// Mitsubishi GX Works2 project: CydeusPlatform3   PLC: FX3U/FX3UC

TYPE ST_1SolCylinderInterface : STRUCT
  bBusy : BOOL;
  bError : BOOL;
  bDone : BOOL;
  bGoActive : BOOL;
  bReset : BOOL;
  tDelayTime : TIME;
  tTimeout : TIME;
  bAbort : BOOL;
END_STRUCT END_TYPE

TYPE ST_ServoMotorInterface : STRUCT
  bBusy : BOOL;
  bError : BOOL;
  bDone : BOOL;
  bServoEnabled : BOOL;
  bEnable : BOOL;
  bStop : BOOL;
  bAbort : BOOL;
  bReset : BOOL;
  bJogPos : BOOL;
  bJogNeg : BOOL;
  bMoveRel : BOOL;
  rMoveDist : REAL;
  rMoveVel : REAL;
  rMoveAccel : REAL;
  rJogVel : REAL;
END_STRUCT END_TYPE

// global labels: GVL_Error
VAR_GLOBAL
  arrError AT M200 : ARRAY [0..9] OF BOOL;  (* List of Current active error *)
END_VAR
VAR_GLOBAL CONSTANT
  uiNumErrMinus1 : INT := 9;  (* Maximum error minus 1 *)
END_VAR
VAR_GLOBAL
  arrMsg AT M250 : ARRAY [0..9] OF BOOL;  (* List of Current active message *)
END_VAR
VAR_GLOBAL CONSTANT
  uiNumMsgMinus1 : INT := 9;  (* Maximum message minus 1 *)
END_VAR

// global labels: GVL_Main
VAR_GLOBAL
  bAlarmTrigger : BOOL;  (* Simulating Alarm Trigger *)
  bMachineError AT M100 : BOOL;  (* Machine error *)
  bManualMode : BOOL;  (* Manual Mode on *)
  bAutoMode : BOOL;  (* Automatic Mode on *)
  bStepMode : BOOL;  (* Step Mode on *)
  bSimMode : BOOL;  (* Simulation Mode on *)
  objPunching : CL_1Sol1SenCylinder;  (* Punching object *)
  stServoMotor : ST_ServoMotorInterface;  (* Servo Motor interface struct *)
  stPunching : ST_1SolCylinderInterface;  (* Punching interface struct *)
  objServoMotor : CL_ServoMotor;  (* Servo Motor object *)
  bManualEnable : BOOL;  (* Manual Mode enabled *)
  bMachineReady AT M101 : BOOL;  (* Machine Ready *)
END_VAR

// global labels: GVL_HMI
VAR_GLOBAL
  btnInitialize AT M2 : BOOL;  (* Begin button *)
  btnAutoMode AT M4 : BOOL;  (* Automatic Mode button *)
  btnStepMode AT M5 : BOOL;  (* Step Mode button *)
  btnTest AT M7 : BOOL;  (* Test Mode button *)
  btnTestManualOn AT M8 : BOOL;  (* Manual Mode Trigger button *)
  btnSetup AT M9 : BOOL;  (* Setup Mode button *)
  btnStartAuto AT M11 : BOOL;  (* Automatic Mode Start button *)
  tboxPulsePerRev AT D200 : REAL;  (* Pulse per revolution textbox *)
  tboxRadius AT D202 : REAL;  (* Radius textbox *)
  tboxMoveVel AT D204 : REAL;  (* Relative Move velocity textbox *)
  tboxMoveAccel AT D206 : DINT;  (* Relative Move accelleration time textbox *)
  tboxPunchingDelayTime AT D210 : DINT;  (* Punching delay time textbox *)
  tboxPunchingTimeout AT D212 : DINT;  (* Punching timeout textbox *)
  btnServoStop AT M14 : BOOL;  (* Servo Stop button *)
  btnServoEnable AT M13 : BOOL;  (* Servo Enable button *)
  btnServoAbort AT M15 : BOOL;  (* Servo Abort button *)
  btnServoReset AT M16 : BOOL;  (* Servo Reset button *)
  btnServoJogPos AT M17 : BOOL;  (* Servo Positive Jog button *)
  btnServoJogNeg AT M18 : BOOL;  (* Servo Negative Jog button *)
  btnServoMoveRel AT M19 : BOOL;  (* Servo Relative Move button *)
  tboxMoveDist AT D126 : REAL;  (* Relative Move distance textbox *)
  btnNextStep AT M6 : BOOL;  (* Next step button *)
  btnStopAuto AT M12 : BOOL;  (* Automatic Mode Stop button *)
  btnLanguage AT D500 : INT;  (* Language selection textbox *)
  btnPunchingOutput AT M20 : BOOL;  (* Punching Active button *)
  btnPunchingReset AT M21 : BOOL;  (* Punching Reset button *)
  btnManualMode AT M3 : BOOL;  (* Manual Mode button *)
  btnAbort AT M0 : BOOL;  (* Abort button *)
  btnReset AT M1 : BOOL;  (* Reset button *)
  btnBack AT M10 : BOOL;  (* Back button *)
  tboxProductLength AT D218 : INT;  (* Product length textbox *)
  tboxNumProduct AT D219 : INT;  (* Product number textbox *)
  btnRunContinuous AT M22 : BOOL;  (* Automatic Mode Continuous Run button *)
  btnClearBatchCounter AT M23 : BOOL;  (* Clear batch counter button *)
  tboxCycleTime AT D122 : REAL;  (* Cycle time textbox *)
  btnManualOutput AT M24 : BOOL;  (* Manual Output control button *)
  btnMaPunchingOutput AT M25 : BOOL;  (* Manual Punching active button *)
  btnMaServoPP AT M26 : BOOL;  (* Manual Servo PP button *)
  btnMaServoNP AT M27 : BOOL;  (* Manual Servo NP button *)
  btnMaServoEM2 AT M28 : BOOL;  (* Manual Servo EM2 button *)
  btnMaServoSON AT M29 : BOOL;  (* Manual Servo SON button *)
  btnMaServoRES AT M30 : BOOL;  (* Manual Servo RES button *)
  tboxCurrentProduct AT D130 : INT;  (* Current product counter textbox *)
  btnInitialPunch AT M31 : BOOL;  (* First Spare material cutting button *)
  tboxRatio AT D214 : REAL;  (* Ratio textbox *)
  btnServoMoveInverse AT M32 : BOOL;  (* Servo Inverse Move button *)
  tboxJogVel AT D216 : REAL;  (* Jog Velocity textbox *)
  btnMaBuzzer AT M33 : BOOL;  (* Manual Buzzer button *)
  tboxOffset AT D220 : REAL;  (* Offset textbox *)
END_VAR

// global labels: GVL_Output
VAR_GLOBAL
  boPunchingOutput AT Y006 : BOOL;  (* Physical output Punching activation *)
  bAuPunchingOutput : BOOL;  (* Software output Punching activation *)
  boServoPP AT Y000 : BOOL;  (* Physical output Servo PP *)
  boServoNP AT Y001 : BOOL;  (* Physical output Servo NP *)
  boServoSON AT Y004 : BOOL;  (* Physical output Servo SON *)
  boServoRES AT Y005 : BOOL;  (* Physical output Servo RES *)
  boServoEM2 AT Y003 : BOOL;  (* Physical output Servo EM2 *)
  bAuServoPP : BOOL;  (* Software output Servo PP *)
  bAuServoNP : BOOL;  (* Software output Servo NP *)
  bAuServoSON : BOOL;  (* Software output Servo SON *)
  bAuServoRES : BOOL;  (* Software output Servo RES *)
  bAuServoEM2 : BOOL;  (* Software output Servo EM2 *)
  boBuzzer AT Y007 : BOOL;  (* Physical output Buzzer *)
  bAuBuzzer : BOOL;  (* Software output Buzzer *)
END_VAR

// global labels: GVL_Input
VAR_GLOBAL
  biEstop1 AT X000 : BOOL;  (* Physical input Emergency Stop 1 *)
  biEstop2 AT X001 : BOOL;  (* Physical input Emergency Stop 2 *)
  biPunchingDone AT X002 : BOOL;  (* Physical input Punching done *)
  biFeederSensor AT X003 : BOOL;  (* Physical input Feeder Sensor *)
  biServoINP AT X005 : BOOL;  (* Physical input Servo INP *)
  biServoRD AT X006 : BOOL;  (* Physical input Servo RD *)
  biServoALM AT X007 : BOOL;  (* Physical input Servo ALM *)
  bEstop1 : BOOL;  (* Software input Emergency Stop 1 *)
  bEstop2 : BOOL;  (* Software input Emergency Stop 2 *)
  bPunchingDone : BOOL;  (* Software input Punching done *)
  bFeederSensor : BOOL;  (* Software input Feeder Sensor *)
  bServoINP : BOOL;  (* Software input Servo INP *)
  bServoRD : BOOL;  (* Software input Servo RD *)
  bServoALM : BOOL;  (* Software input Servo ALM *)
  biStartButton AT X004 : BOOL;  (* Physical input Start button *)
  bStartButton : BOOL;  (* Software input Start button *)
END_VAR

// global labels: GVL_System
VAR_GLOBAL
  bCommandComplete AT M8029 : BOOL;  (* Servo run command completed *)
END_VAR

// global labels: GVL_StateMachine
VAR_GLOBAL
  bInitializingDone : BOOL;  (* Initializing Done *)
  bInitializingAbort : BOOL;  (* Initializing Aborted *)
  iStateInit : INT;  (* Initializing state machine state counter *)
  iStateAuto AT D103 : INT;  (* Automatic mode state machine state counter *)
  bAutoModeDone : BOOL;  (* Automatic mode done *)
  bStopAutoHold : BOOL;  (* Hold stop signal *)
  bAbortDone : BOOL;  (* Abort procedure busy *)
  iStateGeneral AT D100 : INT;  (* General state machine state counter *)
  iLastState AT D101 : INT;  (* Last state temporary variable *)
  bResetBusy : BOOL;  (* Reset procedure busy *)
  bAutoModeStarted AT M120 : BOOL;  (* Automatic mode started *)
  iStateTest AT D102 : INT;  (* Test mode state machine state counter *)
  bManualModeReset : BOOL;  (* Manual mode reset *)
  iCurrentProduct : INT;  (* Current cutted product counter *)
  tonCycleTime : TON;  (* Cycle time timer *)
  rCycleTime : REAL;  (* Cycle time *)
  tpBuzzer : TP;  (* Buzzer active timer *)
  bCompleteBatch : BOOL;  (* Batch completed *)
END_VAR

// task Task_01 (event TRUE, interval 0, priority 31): MAIN

PROGRAM MAIN
VAR
  fbErrorController : FB_ErrorController;
  fbOutputController : FB_OutputController;
  fbStateMachine : FB_StateMachine;
  fbInputLinker : FB_InputLinker;
  fbObjectExecution : FB_ObjectExecution;
END_VAR

(*Input Linker*)
fbInputLinker();

(*State Machine*)
fbStateMachine();

(*Object Execution*)
fbObjectExecution();

(*Output Controller*)
fbOutputController();

(*Error Controller*)
fbErrorController(bResetError := btnReset);
bMachineError := fbErrorController.bError;
END_PROGRAM

FUNCTION_BLOCK FB_ErrorController
VAR
  ii : INT;
END_VAR
VAR_OUTPUT
  bError : BOOL;  (* Error output *)
END_VAR
VAR_INPUT
  bResetError : BOOL;  (* Reset error *)
END_VAR
(*Error Controller - Control errors displayed on HMI*)

(*Reset Errors*)
IF bResetError THEN
	FOR ii := 0 TO uiNumErrMinus1  DO
		arrError[ii] := FALSE;
	END_FOR;
END_IF;

(*Register Errors*)
SET(bAlarmTrigger, arrError[0]);
SET(stPunching.bError, arrError[1]);
SET(stServoMotor.bError, arrError[2]);
SET(NOT bEstop1, arrError[3]);
SET(NOT bEstop2, arrError[4]);

(*Machine Error Trigger*)
bError := FALSE;
FOR ii := 0 TO uiNumErrMinus1  DO
	bError := bError OR arrError[ii];
END_FOR;

(*Register Messages*)
arrMsg[0] := NOT bFeederSensor;
arrMsg[1] := bAutoMode;
arrMsg[2] := bManualMode;
arrMsg[3] := bStepMode;
arrMsg[4] := btnTestManualOn;
arrMsg[5] := bMachineReady;
arrMsg[6] := bInitializingAbort;
END_FUNCTION_BLOCK

FUNCTION FUN_Output
VAR_INPUT
  b_OutAuto : BOOL;
  b_OutMan : BOOL;
  b_ManualMode : BOOL;
END_VAR
(* Output manual and automatic switch*)

FUN_Output := (b_ManualMode AND b_OutMan) OR (NOT b_ManualMode AND b_OutAuto);
END_FUNCTION

FUNCTION_BLOCK FB_OutputController
(*Output Controller - Control automatic and manual output*)

(*Hold current status of output*)
IF LDP(TRUE, btnManualOutput) THEN
		btnMaPunchingOutput := boPunchingOutput ;
		btnMaServoEM2 := boServoEM2;
		btnMaServoNP := boServoNP;
		btnMaServoPP := boServoPP;
		btnMaServoRES := boServoRES;
		btnMaServoSON := boServoSON;
		btnMaBuzzer := boBuzzer;
END_IF;

(*Calculate the logical output, choose auto or man output to be applied, then assign to physical output*)
boPunchingOutput := FUN_Output(btnManualOutput, bAuPunchingOutput, btnMaPunchingOutput);
boServoEM2:= FUN_Output(btnManualOutput, bAuServoEM2, btnMaServoEM2);
boServoNP:= FUN_Output(btnManualOutput, bAuServoNP, btnMaServoNP);
boServoPP:= FUN_Output(btnManualOutput, bAuServoPP, btnMaServoPP);
boServoRES:= FUN_Output(btnManualOutput, bAuServoRES, btnMaServoRES);
boServoSON:= FUN_Output(btnManualOutput, bAuServoSON, btnMaServoSON);
boBuzzer:= FUN_Output(btnManualOutput, bAuBuzzer, btnMaBuzzer);
END_FUNCTION_BLOCK

FUNCTION_BLOCK FB_ManualMode
VAR
  arrTempHold : ARRAY [0..9] OF BOOL;  (* Hold state of outputs *)
END_VAR
VAR CONSTANT
  iTempHoldSize : INT := 9;  (* Size of state holding array *)
END_VAR
VAR
  ii : INT;
END_VAR
(*Manual Mode*)

(* Reset temporary variable state when abort *)
IF bManualModeReset THEN
		FOR ii := 0 TO iTempHoldSize DO 
			arrTempHold[ii] := FALSE;
		END_FOR;
END_IF;


IF (iStateGeneral = 60) OR (iStateGeneral = 100) THEN
		(*Enable Manual Mode*)
		bManualEnable := btnTestManualOn OR (iStateGeneral = 60);
		
		(*Hold Current status of Outputs*)
		IF LDP(TRUE, bManualEnable) THEN
			btnServoAbort := stServoMotor.bAbort;
			btnServoEnable := stServoMotor.bEnable;
			btnServoStop := stServoMotor.bStop;
			btnServoReset := stServoMotor.bReset OR btnReset;
			btnServoJogPos := stServoMotor.bJogPos;
			btnServoJogNeg := stServoMotor.bJogNeg;
			btnServoMoveRel := stServoMotor.bMoveRel;

			btnPunchingOutput := FALSE;
			btnPunchingReset := stPunching.bReset OR btnReset;
			
			arrTempHold[0] := stServoMotor.bAbort;
			arrTempHold[1] := stServoMotor.bEnable;
		END_IF;
		
		(*Restore status to output*)
		IF LDF(TRUE, bManualEnable ) THEN
			stServoMotor.bAbort := arrTempHold[0];
			stServoMotor.bEnable := arrTempHold[1];
		END_IF;
				
		(*Buttons on HMI control servo motor and punching*)
		IF bManualEnable THEN
			stServoMotor.bAbort := btnServoAbort;
			stServoMotor.bEnable := btnServoEnable;
			stServoMotor.bStop := btnServoStop;
			stServoMotor.bReset := btnServoReset OR btnReset;
			stServoMotor.bJogPos := btnServoJogPos;
			stServoMotor.bJogNeg := btnServoJogNeg;
			stServoMotor.rJogVel := tboxJogVel;
			stServoMotor.bMoveRel := btnServoMoveRel;
			IF btnServoMoveInverse THEN
					stServoMotor.rMoveDist := -(tboxMoveDist + tboxOffset);
			ELSE
					stServoMotor.rMoveDist := tboxMoveDist + tboxOffset;
			END_IF;
			
			stPunching.bGoActive := btnPunchingOutput;
			stPunching.bReset := btnPunchingReset OR btnReset;
			stPunching.bAbort := btnPunchingReset;
		END_IF;
END_IF;
END_FUNCTION_BLOCK

FUNCTION_BLOCK FB_Initializing
VAR
  fbDelayStep0 : TON;  (* Step 0 delay timer *)
  fbDelayStep10 : TON;  (* Step 10 delay timer *)
END_VAR
(*Initializing*)

IF iStateGeneral = 20 THEN
		(*State Machine*)
		CASE iStateInit OF
				0: 	(*Home the punching*)
						IF stPunching.bDone OR fbDelayStep0.Q THEN
								iStateInit := 10;
						END_IF;
						
				10:	(*Spare state*)
						IF (*stServoMotor.bServoEnabled*) TRUE THEN
								iStateInit := 20;
						ELSIF fbDelayStep10.Q THEN
								iStateInit := 50;
						END_IF;
						
				20: 	(*Done*)
						;
				50: 	(*Abort*)	
						;
		END_CASE;
		
		(*State Action*)
		RST((iStateInit = 0), stPunching.bGoActive);
		SET((iStateInit = 10), stServoMotor.bEnable);
		
		bInitializingDone := iStateInit = 20;									(* Initializing done signal *)
		bInitializingAbort := iStateInit = 50;									(* Initializing abort signal *)
END_IF;

(*Function block call*)
fbDelayStep0(IN := iStateInit = 0 AND NOT fbDelayStep0.Q, PT := t#2s);
fbDelayStep10(IN := iStateInit = 10 AND NOT fbDelayStep10.Q, PT := t#5s);
END_FUNCTION_BLOCK

FUNCTION_BLOCK FB_StateMachine
VAR
  fbInitializing : FB_Initializing;  (* Initializing action *)
  fbAutoMode : FB_AutoMode;  (* Automatic action *)
  fbManualMode : FB_ManualMode;  (* Manual action *)
  fbAborting : FB_Aborting;  (* Abort action *)
  fbReset : FB_Reset;  (* Reset action *)
END_VAR
(*Main State Machine*)

(*Abort command*)
IF (btnAbort OR bMachineError OR NOT bEstop1 OR NOT bEstop2) AND NOT (iStateGeneral = 10) AND NOT (iStateGeneral >= 100) THEN	
	iStateGeneral := 0;
END_IF;

(*Reset command*)
IF btnReset  OR bResetBusy THEN
	fbReset();
END_IF;

(*Main state machine*)
CASE iStateGeneral OF
	0: 		(*Aborting*)
		IF bAbortDone THEN
			iStateGeneral := 10;
		END_IF;
	
	10: 		(*Begin*)
		IF btnInitialize AND NOT bMachineError THEN
			iStateGeneral := 20;
		ELSIF btnTest THEN
			iLastState := iStateGeneral;
			iStateGeneral := 100;
		ELSIF btnSetup THEN
			iLastState := iStateGeneral;
			iStateGeneral := 150;
		END_IF;
		
	20: 		(*Initializing*)
		IF bInitializingDone AND NOT bMachineError THEN
			iStateGeneral := 30;
		END_IF;
		
	30: 		(*Ready*)
		IF btnAutoMode AND NOT bMachineError THEN
			iStateGeneral := 40;
		ELSIF btnStepMode AND NOT bMachineError THEN
			iStateGeneral := 50;
		ELSIF btnManualMode AND NOT bMachineError THEN
			iStateGeneral := 60;
		ELSIF btnTest THEN
			iLastState := iStateGeneral;
			iStateGeneral := 100;
		END_IF;
	
	40: 		(*Running Auto Mode*)
		IF btnBack OR bAutoModeDone  AND NOT bMachineError THEN
			iStateGeneral := 30;
		END_IF;
		
	50: 		(*Running Step Mode*)
		IF btnBack OR bAutoModeDone AND NOT bMachineError THEN
			iStateGeneral := 30;
		END_IF;
		
	60: 		(*Running Manual Mode*)
		IF btnBack AND NOT bMachineError THEN
			iStateGeneral := 30;
		END_IF;
		
	100: 		(*Testing*)
		IF btnBack THEN
			iStateGeneral := iLastState;
		END_IF;
		
	150: 		(*Setting*)
		IF btnBack THEN
			iStateGeneral := iLastState;
		END_IF;
	
ELSE 
		;
END_CASE;

(*State Action*)
bAutoMode := iStateGeneral = 40;																	(*In Automatic Mode*)
bStepMode := iStateGeneral = 50;																	(*In Step Mode*)
bManualMode := iStateGeneral = 60;																(*In Manual Mode*)
bMachineReady := (iStateGeneral >= 30) AND (iStateGeneral < 100);	(*Machine Ready signal*)
IF LDP(TRUE, iStateGeneral = 100) THEN													(*Reset test mode state machine*)
		iStateTest := 0;
END_IF;	

stServoMotor.bEnable := (iStateGeneral >= 40) AND (iStateGeneral <= 60);	(*Enable servo motor when ready*)
tpBuzzer(IN := bAutoModeDone OR bCompleteBatch OR tpBuzzer.Q, pt:= t#5s);	
bAuBuzzer := tpBuzzer.Q;																						(*Buzzer activated when batch done*)

		(*Clear product counter*)
		IF btnClearBatchCounter OR bStartButton THEN
				iCurrentProduct := 0;
				tboxCurrentProduct := 0;
				tboxCycleTime := 0.0;
		END_IF;

(*Function Block Call*)
bInitializingDone := FALSE;
bInitializingAbort := FALSE;
bAutoModeDone := FALSE;
bAbortDone := FALSE;
bAutoModeStarted := FALSE;
bCompleteBatch := FALSE;

fbAborting();
fbInitializing();
fbAutoMode(bEnStepMode := iStateGeneral = 50, bNext := btnNextStep);
fbManualMode();
END_FUNCTION_BLOCK

FUNCTION_BLOCK FB_AutoMode
VAR_INPUT
  bEnStepMode : BOOL;  (* Enable step mode *)
  bNext : BOOL;  (* Go to next step signal *)
END_VAR
VAR
  bNextStep : BOOL;  (* Next step variable *)
  bExit : BOOL;  (* Exit from automode *)
  bDelayState : BOOL;  (* Delay state signal *)
  tonDelayState : TON;  (* Delay state timer *)
END_VAR
IF iStateGeneral = 40 OR iStateGeneral = 50 THEN
		(*Auto Mode State Machine*)
		CASE iStateAuto OF
				0: 		(*Ready*)
						IF btnStartAuto OR bStartButton THEN
							iStateAuto := 10;
						END_IF;
						
				10: 		(*Wait for raw material*)
						IF bFeederSensor AND bNextStep THEN
							iStateAuto := 15;
						END_IF;
						
				15:		(*Check if Initial punch needed*)
						IF btnInitialPunch THEN
							iStateAuto := 20;
						ELSE
							iStateAuto := 30;
						END_IF;
						
				20: 		(*Cut spare material before beginning*)
						IF stPunching.bDone AND bNextStep THEN
							iStateAuto := 30;
						END_IF;
						
				30: 		(*Set parameters*)
						bDelayState := NOT bDelayState;
						IF NOT btnServoMoveInverse THEN
							stServoMotor.rMoveDist := INT_TO_REAL(tboxProductLength) + tboxOffset;	
						ELSE
							stServoMotor.rMoveDist := -(INT_TO_REAL(tboxProductLength) + tboxOffset);							
						END_IF;	
						IF bDelayState THEN
							iStateAuto := 40;
						END_IF;
				
				40: 		(*Feed new raw material to punching machine*)
						IF stServoMotor.bDone AND bNextStep THEN
							iStateAuto := 50;
						END_IF;
					
				50: 		(*Cut raw material into final product*)
						IF stPunching.bDone AND bNextStep THEN
							iStateAuto := 60;
						END_IF;
						
				60: 		(*Count a completed product*)
						iCurrentProduct := iCurrentProduct + 1;
						iStateAuto := 70;
		
				70: 		(*Check for raw material or stop button pressed*)
						IF (NOT bFeederSensor OR (iCurrentProduct >= tboxNumProduct AND NOT btnRunContinuous)) AND NOT bStopAutoHold THEN
							iStateAuto := 75;
						ELSIF bFeederSensor AND NOT bStopAutoHold THEN
							iStateAuto := 30;
						ELSIF bStopAutoHold THEN 
							iStateAuto := 100;
						END_IF;
						
				75: 		(*Complete a batch*)
						IF tonDelayState.Q THEN
							iStateAuto := 100;
						END_IF;
						
				80: 		(*Auto mode done*)
						;
						
				100: 	(*Stop procedure*)
						IF btnStartAuto OR bStartButton THEN
							iStateAuto := 30;
						ELSIF bExit THEN 
							iStateAuto := 80;
						END_IF;
						
		END_CASE;
		
		(*Auto Mode State Action*)
		bNextStep := (NOT bEnStepMode OR (bEnStepMode AND bNext));		(* Button next step pressed *)
		SET(btnStopAuto, bStopAutoHold);															(* Hold stop button *)
		RST(iStateAuto = 100, bStopAutoHold);
		bAutoModeDone:= iStateAuto = 80;															(* Auto mode done signal *)
		bCompleteBatch := iStateAuto = 75;															(* Batch completed signal *)
		bAutoModeStarted := iStateAuto >= 10 AND iStateAuto < 100;			(* Auto mode started signal *)
		
		stServoMotor.bMoveRel := (iStateAuto = 40);											(* Servo moving condition *)
		stPunching.bGoActive := (iStateAuto = 20) OR (iStateAuto = 50);		(* Punching moving condition *)
		
ELSIF iStateGeneral = 30 THEN																			(* Reset state machine when in ready *)
		iStateAuto := 0;
		bStopAutoHold := FALSE;
END_IF;

(*Cycle time calculation*)
IF (iStateAuto = 60) OR  (iStateAuto = 70) THEN
		tboxCycleTime := rCycleTime;
		tboxCurrentProduct := iCurrentProduct;
END_IF;

IF iStateAuto = 30 THEN
		rCycleTime := 0.0;
END_IF;

tonCycleTime(IN := NOT tonCycleTime.Q AND ((iStateAuto = 40) OR (iStateAuto = 50)), PT := t#100ms);
IF tonCycleTime.Q THEN
		rCycleTime := rCycleTime + 0.1;
END_IF;

tonDelayState(in := (iStateAuto = 75), pt := t#100ms);
END_FUNCTION_BLOCK

FUNCTION_BLOCK FB_InputLinker
(*Input Linker*)

(*Link physical input to logical input memory*)
IF NOT bSimMode THEN	
		bEstop1 := biEstop1;
		bEstop2 := biEstop2;
		bFeederSensor := biFeederSensor;
		bPunchingDone := biPunchingDone;
		bServoINP := biServoINP;
		bServoRD := biServoRD;
		bServoALM := biServoALM;
		bStartButton := biStartButton;
END_IF;
END_FUNCTION_BLOCK

FUNCTION_BLOCK FB_ObjectExecution
VAR
  tboxRatioInt : DINT;
END_VAR
(* Object excution - Execute the servo and punching object *)

(* Limit the servo speed *)
IF (tboxMoveVel*tboxRatio) > 3000.0 THEN
		tboxMoveVel := 3000.0/tboxRatio;
END_IF;		
IF (tboxJogVel*tboxRatio) > 3000.0 THEN
		tboxJogVel := 3000.0/tboxRatio;
END_IF;	

(* Pass parameter and execute servo *)
objServoMotor(biINP := bServoINP,
								biRD := bServoRD,
								biALM := bServoALM,
								boNPz := bAuServoNP,
								boEM2 := bAuServoEM2,
								boRES := bAuServoRES,
								boSON := bAuServoSON,
								
								bEnable := stServoMotor.bEnable,
								bStop := stServoMotor.bStop,
								bAbort := stServoMotor.bAbort,
								bReset := stServoMotor.bReset,
								iOutChannel := 0,
								iMoveDelay := 100,
								rPulsePerRev := tboxPulsePerRev,
								rRadius := tboxRadius,
								rRatio := tboxRatio,
								
								bJogPos := stServoMotor.bJogPos,
								bJogNeg := stServoMotor.bJogNeg,
								iJogVel := (tboxJogVel*tboxRatio),
								
								bMoveRel := stServoMotor.bMoveRel,
								rMoveDist := stServoMotor.rMoveDist,
								iMoveVel := (tboxMoveVel*tboxRatio),
								iMoveAccel := tboxMoveAccel,

								bBusy := stServoMotor.bBusy,
								bDone := stServoMotor.bDone,
								bError := stServoMotor.bError,
								bServoEnabled := stServoMotor.bServoEnabled);
								

(* Pass parameter and execute punching *)								
objPunching(biSensorDone := bPunchingDone,
							biActiveFeedback := bAuPunchingOutput,
							boSolenoid := bAuPunchingOutput,
							
							bAbort := stPunching.bAbort,
							bGoActive := stPunching.bGoActive,
							bReset := stPunching.bReset,
							tDelayTime := tboxPunchingDelayTime,
							tTimeout := tboxPunchingTimeout,

							bBusy := stPunching.bBusy,
							bDone := stPunching.bDone,
							bError := stPunching.bError);
END_FUNCTION_BLOCK

FUNCTION_BLOCK CL_1Sol1SenCylinder
VAR_INPUT
  biSensorDone : BOOL;  (* Sensor done input *)
  bGoActive : BOOL;  (* Go active command *)
  bReset : BOOL;  (* Reset command *)
END_VAR
VAR_OUTPUT
  boSolenoid : BOOL;  (* Coil active output *)
  bBusy : BOOL;  (* Busy output *)
  bInHomePos : BOOL;  (* In home position output *)
  bError : BOOL;  (* Error output *)
END_VAR
VAR_INPUT
  tDelayTime : DINT;  (* Delay time parameter *)
  tTimeout : DINT;  (* Time out parameter *)
END_VAR
VAR
  fbDelayTime : TP;  (* Delay timer *)
  fbTimeout : TON;  (* Timeout timer *)
END_VAR
VAR_INPUT
  biActiveFeedback : BOOL;  (* Coil active feedback signal *)
END_VAR
VAR
  bSensorDoneHold : BOOL;  (* Hold sensor done signal *)
  tDelay : TIME;  (* Delay time (Type Time) *)
  tTimeoutz : TIME;  (* Timeout (Type Time) *)
END_VAR
VAR_OUTPUT
  bDone : BOOL;  (* Done output *)
END_VAR
VAR_INPUT
  bAbort : BOOL;  (* Abort command *)
END_VAR
VAR
  bActivating : BOOL;  (* Cylinder active signal *)
END_VAR
(* Cylinder class, use for cylinder with 1 limit sensor and 1 coil *)


(*Activate Output: Enable solenoid on valve when going active command raised*) 
boSolenoid := LDP(TRUE, bGoActive) OR boSolenoid AND NOT fbTimeout.Q AND NOT LDP(TRUE, biSensorDone);

(*Process Input: If sensor done signal was caught, command is done*)
SET(LDP(TRUE, biSensorDone), bSensorDoneHold);							(* Wait for sensors signal *)
RST(LDP(TRUE, bBusy), bSensorDoneHold);											(* Reset when done *)
bInHomePos := NOT fbDelayTime.Q AND bSensorDoneHold;			(* After sensor done raised, timer will count and wait for stable position *)
bBusy := bActivating OR fbDelayTime.Q;													(* Cylinder is busy when activating or waiting for stable *)
bActivating:= biActiveFeedback AND boSolenoid AND NOT LDP(TRUE, biSensorDone); 	
bDone := NOT bBusy AND NOT bActivating AND bGoActive;			(* Cylinder is done if not busy *)

(*Error handling*)
		(*Notify timeout error*)
		SET(fbTimeout.Q, bError);

		(*Reset timeout error*)
		RST(bReset, bError);
		
(*Abort*)
IF bAbort THEN
		boSolenoid := FALSE;
		bSensorDoneHold := TRUE;
END_IF;

(*Timers call*)
tDelay := DINT_TO_TIME(tDelayTime);
tTimeoutz := DINT_TO_TIME(tTimeout);
fbDelayTime(IN := LDF(TRUE, bActivating) OR fbDelayTime.Q, PT := tDelay );
fbTimeout(IN := bBusy, PT := tTimeoutz );
END_FUNCTION_BLOCK

FUNCTION_BLOCK FB_Aborting
VAR
  fbAbortHold : TP;
END_VAR
(*Aborting*)

IF iStateGeneral = 0 THEN
		(*Abort object*)
		stServoMotor.bEnable := FALSE;							(* Disable servo *)
		stServoMotor.bAbort := fbAbortHold.Q;					(* Abort servo *)
		stServoMotor.bStop := FALSE;								(* Disable command *)
		stServoMotor.bJogNeg := FALSE;
		stServoMotor.bJogPos := FALSE;
		stServoMotor.bMoveRel := FALSE;
		
		stPunching.bGoActive := FALSE;							(* Disable cylinder *)
		stPunching.bAbort := fbAbortHold.Q;						(* Abort cylinder*)
		
		(*About function block*)
		bManualModeReset := fbAbortHold.Q;
		
		(*Clear variables*)
		iStateInit := 0;
		iStateAuto := 0;
		bStopAutoHold := FALSE;
		iCurrentProduct := 0;
		rCycleTime := 0.0;
		
		bAbortDone := NOT btnAbort AND NOT fbAbortHold.Q;
END_IF;

fbAbortHold(IN := btnAbort OR fbAbortHold.Q, PT := t#1000ms);
END_FUNCTION_BLOCK

FUNCTION_BLOCK FB_Reset
(* Reset *)

(* Reset all objects *)
stPunching.bReset := btnReset;
stServoMotor.bReset := btnReset;
bResetBusy := btnReset;							(* Reset busy signal *)
END_FUNCTION_BLOCK

FUNCTION_BLOCK CL_ServoMotor
VAR_INPUT
  biINP : BOOL;  (* Servo INP input *)
  biRD : BOOL;  (* Servo RD input *)
  biALM : BOOL;  (* Servo ALM input *)
  bEnable : BOOL;  (* Enable command *)
  bStop : BOOL;  (* Stop command *)
  bAbort : BOOL;  (* Abort command *)
  bReset : BOOL;  (* Reset command *)
  bJogPos : BOOL;  (* Positive Jog command *)
  bJogNeg : BOOL;  (* Negative Jog command *)
  bMoveRel : BOOL;  (* Move Relative command *)
  rMoveDist : REAL;  (* Move distance parameter *)
END_VAR
VAR_OUTPUT
  boEM2 : BOOL;  (* Servo EM2 output *)
  boSON : BOOL;  (* Servo SON output *)
  boRES : BOOL;  (* Servo RES output *)
  bBusy : BOOL;  (* Busy output *)
  bError : BOOL;  (* Error output *)
  bDone : BOOL;  (* Done output *)
  bServoEnabled : BOOL;  (* Servo Enabled output *)
END_VAR
VAR
  iState : INT;  (* State machine state counter *)
  fbResetHold : TP_10;  (* Reset command holding timer *)
  bResetHold : BOOL;  (* Hold reset command *)
  fbMoveDelay : TON;  (* Move delay timer *)
END_VAR
VAR_INPUT
  iMoveDelay : WORD;  (* Moving delay time *)
END_VAR
VAR
  tMoveDelay : TIME;  (* Move delay time *)
  iStopState : INT;  (* Stopping state machine state counter *)
END_VAR
VAR_INPUT
  iMoveVel : REAL;  (* Move velocity parameter *)
  iMoveAccel : DINT;  (* Move accelleration parameter *)
  rPulsePerRev : REAL;  (* Pulse per revolution parameter *)
  rRadius : REAL;  (* Roller radius parameter *)
END_VAR
VAR
  iFrequency : DINT;  (* Output pulse frequency *)
  iPulse : DINT;  (* Output pulse number *)
  iAccel : DINT;  (* Output pulse accelleration time *)
  bOutPulse : BOOL;  (* Output pulse trigger *)
END_VAR
VAR_INPUT
  iOutChannel : INT;  (* Pulse Output channel selection *)
END_VAR
VAR
  bInCommand : BOOL;  (* In command variable *)
  bCompleted : BOOL;  (* Completed variable *)
  tonDelayComplete : TON_10;  (* Complete delay timer *)
  bCompletedHold : BOOL;  (* Hold Complete signal *)
END_VAR
VAR_OUTPUT
  boNPz : BOOL;  (* Servo NP output *)
END_VAR
VAR_INPUT
  rRatio : REAL;  (* Gear ratio parameter *)
  iJogVel : REAL;  (* Jog velocity parameter *)
END_VAR
(* Motor class, use for servo motor *)

(*Main State Machine*)
CASE iState OF 
		0: 	(*Unenabled, wait for Enable command*)
				IF bEnable AND NOT bStop AND NOT bError THEN
						iState := 10;
				END_IF;
				
		10: 	(*Servo On*)
				IF bServoEnabled THEN
						iState := 20;
				END_IF;
						
		20: 	(*Servo Ready, wait for moving command*)
				IF bJogPos AND NOT bStop AND NOT bError THEN				(* Positive Jog command *)
						iState := 100;
				ELSIF bJogNeg AND NOT bStop AND NOT bError THEN		(* Negative Jog command *)
						iState := 140;
				ELSIF bMoveRel AND NOT bStop AND NOT bError THEN		(* Move Relative command *)
						iState := 200;
				END_IF;
				
		100: 	(*Calculate number of pulse*)			
				iFrequency := REAL_TO_DINT(rPulsePerRev*iJogVel/60.0);
				iPulse := 2147483647;
				iAccel := iMoveAccel;
				iState := 110;
				
		110: 	(*Execute Jog Pos command*)
				IF NOT bJogPos THEN 
						iState := 20;
				END_IF;
				
		140: 	(*Calculate number of pulse*)			
				iFrequency := REAL_TO_DINT(rPulsePerRev*iJogVel/60.0);
				iPulse := 2147483647;
				iAccel := iMoveAccel;
				iState := 150;
				
		150: 	(*Execute Jog Neg command*)
				IF NOT bJogNeg THEN
						iState := 20;
				END_IF;
				
		200: 	(*Calculate number of pulse*)
				iFrequency := REAL_TO_DINT(rPulsePerRev*iMoveVel/60.0);
				iAccel := iMoveAccel;
				tMoveDelay := WORD_TO_TIME(iMoveDelay);
				iState := 210;
				IF rMoveDist > 0.0 THEN
						iPulse := REAL_TO_DINT(rRatio*rPulsePerRev*rMoveDist/(2.0*3.1415926*rRadius));	
				ELSIF rMoveDist < 0.0 THEN
						iPulse := REAL_TO_DINT(rRatio*rPulsePerRev*(-rMoveDist)/(2.0*3.1415926*rRadius));	
				ELSE
						iState := 220;
				END_IF;
		
		210: 	(*Execute Move Relative command*)
				IF tonDelayComplete.Q AND fbMoveDelay.Q THEN		
						iState := 220;
				END_IF;		
				
		220: 	(*Move Relative done, wait for command release*)
				IF NOT bMoveRel THEN
						iState := 20;
				END_IF;
				
END_CASE;
	
(*Procedure*)
		(*Abort command - Reset all state machine*)
		IF bAbort OR NOT bEnable OR bError THEN
				iState := 0;
				iStopState := 0;
		END_IF;
		
		(*Reset command - Reset all state machine*)
		IF bReset AND bError THEN
				iState := 0;
				iStopState := 0;
		END_IF;		
		
		(*Stop command*)
		CASE iStopState OF
				0: 	(*Wait for stop signal*)
						IF bStop THEN
								iStopState := 10;
						END_IF;
						
				10: 	(*Execute Stop*)
						IF iState > 20 THEN
								iState := 20;
						END_IF;
						IF biINP THEN
								iStopState := 20;
						END_IF;
						
				20: 	(*Stop done, wait for command release*)
						IF NOT bStop THEN
								iStopState := 0;
						END_IF;
		END_CASE;	

(*State Action*)
		boSON := (iState >= 10);																			(*Enable Servo Motor*)	
		boEM2 := NOT bAbort AND biALM;													(*Abort Servo Motor*)
		boRES := fbResetHold.Q AND NOT biALM;									(*Reset Servo Motor*)		
		
		bBusy := (iState = 110) OR (iState = 150) OR (iState = 210) OR (iStopState = 10);		(*Servo is busy*)
		bDone := (iState = 220) OR (iStopState = 20);									(*Servo movement is done*)
		bServoEnabled := biRD;																		(*Servo is powered on*)
	
		SET(NOT biALM, bError);																		(*Notify Servo Motor Error*)
		RST((bReset AND bError), bError);													(*Reset object error*)	
		
		bInCommand:= ((iState = 110) OR (iState = 150) OR (iState = 210)) AND NOT (iStopState = 10);	(*Enable Pulse*)
		boNPz := ((iState = 150) OR (rMoveDist < 0.0));												(*Reverse rotation*)
		
		SET(bCompleted, bCompletedHold);
		RST(NOT (iState = 210), bCompletedHold);
		bResetHold := (bReset AND NOT fbResetHold.Q) OR (bResetHold AND fbResetHold.Q) ;
	
(*Function Block Call*)
fbResetHold(IN := bResetHold, PT := t#600ms);
fbMoveDelay(IN := (iState = 210) AND bServoEnabled AND NOT bStop AND NOT bAbort AND NOT bError, PT := tMoveDelay);
tonDelayComplete(IN := biINP AND bCompletedHold, PT:= t#50ms);

(*Output pulse to server drive*)
bOutPulse := (LDP(TRUE, bInCommand) OR bOutPulse) AND NOT (bCompleted AND bMoveRel) AND NOT LDF(TRUE, bInCommand);		(*Output pulse command*)

CASE iOutChannel OF 		(*Choose output channel*)
	0: 	(*Y000*)
			DPLSR(bOutPulse, iFrequency, iPulse, iAccel, Y000);
	1:		(*Y001*)
			DPLSR(bOutPulse, iFrequency, iPulse, iAccel, Y001);
	2:		(*Y002*)
			DPLSR(bOutPulse, iFrequency, iPulse, iAccel, Y002);
END_CASE;
bCompleted := bCommandComplete;
END_FUNCTION_BLOCK
